(* CODESYS project Device.export

Project tree, tasks and I/O mapping:
  Device : CODESYS Control Win V3, 3S - Smart Software Solutions GmbH, version 3.5.17.30
    application Application
      libraries: Standard, * (System); CAA Memory, * (CAA Technical Workgroup); VisuDialogs, * (System); Standard64, * (System); VisuSymbols, 4.1.0.0 (System); Util, * (System); OwenTypes, 3.5.17.5 (Production association OWEN); Mx210 Assistant, 3.5.11.11 (Production association OWEN)
      task MainTask (cyclic, interval t#10ms, priority 1) calls PRG_Main, PRG_HMI
      task VISU_TASK (cyclic, interval 100 ms, priority 31) calls VisuElems.Visu_Prg
      data type E_LevelState
      data type E_WorkMode
      data type ST_ScheduleSlot
      global variables GVL_HMI
      global variables GVL_IO
      global variables GVL_Process
      global variables GVL_Schedules
      global variables TargetVars
      image pool ImagePool
      function block FB_AutoMode [ST]
      function block FB_LevelMonitor [ST]
      function block FB_ManualMode [ST]
      function block FB_Schedule [ST]
      program PRG_HMI [ST]
      program PRG_Main [ST]
      visualisation Visu_Levels
      visualisation Visu_Main
      visualisation Visu_Pumps
      visualisation Visu_Settings
      visualisation Visu_Valves
    Ethernet : Ethernet, 3S - Smart Software Solutions GmbH, version 3.5.17.0
      Modbus_TCP_Master : Modbus TCP Master, 3S - Smart Software Solutions GmbH, version 3.5.17.0
        MV210_214 : MV210-214, Production association OWEN, version 3.5.11.13
            input  Application.SA1_Auto : BOOL  // Битовая маска входов.Вход 1
            input  Application.SA2_Auto : BOOL  // Битовая маска входов.Вход 2
            input  Application.SA3_Auto : BOOL  // Битовая маска входов.Вход 3
            input  Application.SA4_Auto : BOOL  // Битовая маска входов.Вход 4
            input  Application.SA5_Auto : BOOL  // Битовая маска входов.Вход 5
            input  Application.SA6_Auto : BOOL  // Битовая маска входов.Вход 6
            input  Application.LVL_High : BOOL  // Битовая маска входов.Вход 7
            input  Application.LVL_Mid : BOOL  // Битовая маска входов.Вход 8
            input  Application.LVL_Low : BOOL  // Битовая маска входов.Вход 9
            input  Application.Flood : BOOL  // Битовая маска входов.Вход 10
            input  Application.SA7_Auto : BOOL  // Битовая маска входов.Вход 11
            input  Application.SA8_Manual : BOOL  // Битовая маска входов.Вход 12
            input  Application.SA9_Manual : BOOL  // Битовая маска входов.Вход 13
            input  Application.SA10_ManualOpen : BOOL  // Битовая маска входов.Вход 14
            input  Application.SA11_ManualOpen : BOOL  // Битовая маска входов.Вход 15
            input  Application.SA12_ManualOn : BOOL  // Битовая маска входов.Вход 16
            input  Application.SA13_Compressor : BOOL  // Битовая маска входов.Вход 17
            input  Application.DK_QF2 : BOOL  // Битовая маска входов.Вход 18
            input  Application.DK_QF3 : BOOL  // Битовая маска входов.Вход 19
            input  Application.DK_QF4 : BOOL  // Битовая маска входов.Вход 20
            input  Application.DK_QF5 : BOOL  // Битовая маска входов.Вход 21
            input  Application.DK_QF6 : BOOL  // Битовая маска входов.Вход 22
            input  Application.DK_QF7 : BOOL  // Битовая маска входов.Вход 23
            input  Application.DK_QF8 : BOOL  // Битовая маска входов.Вход 24
            input  Application.DK_QF9 : BOOL  // Битовая маска входов.Вход 25
            input  Application.DK_QF10 : BOOL  // Битовая маска входов.Вход 26
            input  Application.DK_QF11 : BOOL  // Битовая маска входов.Вход 27
            input  Application.DK_QF18 : BOOL  // Битовая маска входов.Вход 28
            input  Application.DK_QF19 : BOOL  // Битовая маска входов.Вход 29
            input  Application.DK_QF1 : BOOL  // Битовая маска входов.Вход 30
            unmapped channels: Tmp, Исключить модуль из опроса, Флаг ошибки, Битовая маска входов, Значение счетчика, Значение счетчика, Значение счетчика, Значение счетчика, Значение счетчика, Значение счетчика, Значение счетчика, Значение счетчика, Значение счетчика, Значение счетчика, Значение счетчика, Значение счетчика, Значение счетчика, Значение счетчика, Значение счетчика, Значение счетчика, Значение счетчика, Значение счетчика, Значение счетчика, Значение счетчика, Значение счетчика, Значение счетчика, Значение счетчика, Значение счетчика, Значение счетчика, Значение счетчика, Значение счетчика, Значение счетчика, Значение счетчика, Значение счетчика, Значение счетчика, Значение счетчика, Сбросить счетчик, Сбросить счетчик, Сбросить счетчик, Сбросить счетчик,
              Сбросить счетчик, Сбросить счетчик, Сбросить счетчик, Сбросить счетчик, Сбросить счетчик, Сбросить счетчик, Сбросить счетчик, Сбросить счетчик, Сбросить счетчик, Сбросить счетчик, Сбросить счетчик, Сбросить счетчик, Сбросить счетчик, Сбросить счетчик, Сбросить счетчик, Сбросить счетчик, Сбросить счетчик, Сбросить счетчик, Сбросить счетчик, Сбросить счетчик, Сбросить счетчик, Сбросить счетчик, Сбросить счетчик, Сбросить счетчик, Сбросить счетчик, Сбросить счетчик, Сбросить счетчик, Сбросить счетчик
        MV210_214_1 : MV210-214, Production association OWEN, version 3.5.11.13
            settings: Unit-ID = 2; IPAddress = [192, 168, 0, 2]
            input  Application.VFD1_Run : BOOL  // Битовая маска входов.Вход 1
            input  Application.VFD1_Alarm : BOOL  // Битовая маска входов.Вход 2
            input  Application.VFD2_Run : BOOL  // Битовая маска входов.Вход 3
            input  Application.VFD2_Alarm : BOOL  // Битовая маска входов.Вход 4
            input  Application.FB_KM0 : BOOL  // Битовая маска входов.Вход 5
            input  Application.FB_KM1 : BOOL  // Битовая маска входов.Вход 6
            input  Application.FB_KM2 : BOOL  // Битовая маска входов.Вход 7
            input  Application.FB_KM3 : BOOL  // Битовая маска входов.Вход 8
            input  Application.FB_KM4 : BOOL  // Битовая маска входов.Вход 9
            input  Application.FB_KM5 : BOOL  // Битовая маска входов.Вход 10
            input  Application.FB_KM5_1 : BOOL  // Битовая маска входов.Вход 11
            input  Application.FB_KM6 : BOOL  // Битовая маска входов.Вход 12
            input  Application.FB_KM6_1 : BOOL  // Битовая маска входов.Вход 13
            input  Application.FB_KM7 : BOOL  // Битовая маска входов.Вход 14
            input  Application.FB_KM8 : BOOL  // Битовая маска входов.Вход 15
            input  Application.FB_KM9 : BOOL  // Битовая маска входов.Вход 16
            input  Application.FB_KM10 : BOOL  // Битовая маска входов.Вход 17
            input  Application.FB_KM11 : BOOL  // Битовая маска входов.Вход 18
            input  Application.M2_Closed : BOOL  // Битовая маска входов.Вход 19
            input  Application.M2_Open : BOOL  // Битовая маска входов.Вход 20
            input  Application.M3_Closed : BOOL  // Битовая маска входов.Вход 21
            input  Application.M3_Open : BOOL  // Битовая маска входов.Вход 22
            input  Application.M4_Closed : BOOL  // Битовая маска входов.Вход 23
            input  Application.M4_Open : BOOL  // Битовая маска входов.Вход 24
            input  Application.M5_Closed : BOOL  // Битовая маска входов.Вход 25
            input  Application.M5_Open : BOOL  // Битовая маска входов.Вход 26
            unmapped channels: Tmp, Исключить модуль из опроса, Флаг ошибки, Битовая маска входов, Значение счетчика, Значение счетчика, Значение счетчика, Значение счетчика, Значение счетчика, Значение счетчика, Значение счетчика, Значение счетчика, Значение счетчика, Значение счетчика, Значение счетчика, Значение счетчика, Значение счетчика, Значение счетчика, Значение счетчика, Значение счетчика, Значение счетчика, Значение счетчика, Значение счетчика, Значение счетчика, Значение счетчика, Значение счетчика, Значение счетчика, Значение счетчика, Значение счетчика, Значение счетчика, Значение счетчика, Значение счетчика, Значение счетчика, Значение счетчика, Значение счетчика, Значение счетчика, Сбросить счетчик, Сбросить счетчик, Сбросить счетчик, Сбросить счетчик,
              Сбросить счетчик, Сбросить счетчик, Сбросить счетчик, Сбросить счетчик, Сбросить счетчик, Сбросить счетчик, Сбросить счетчик, Сбросить счетчик, Сбросить счетчик, Сбросить счетчик, Сбросить счетчик, Сбросить счетчик, Сбросить счетчик, Сбросить счетчик, Сбросить счетчик, Сбросить счетчик, Сбросить счетчик, Сбросить счетчик, Сбросить счетчик, Сбросить счетчик, Сбросить счетчик, Сбросить счетчик, Сбросить счетчик, Сбросить счетчик, Сбросить счетчик, Сбросить счетчик, Сбросить счетчик, Сбросить счетчик
        MU210_403 : MU210-403, Production association OWEN, version 3.5.11.13
            settings: Unit-ID = 3; IPAddress = [192, 168, 0, 3]
            output Application.CMD_KM0 : BOOL  // Битовая маска выходов (запись).Выход 1
            output Application.CMD_KM1 : BOOL  // Битовая маска выходов (запись).Выход 3
            output Application.CMD_KM2 : BOOL  // Битовая маска выходов (запись).Выход 4
            output Application.CMD_KM3 : BOOL  // Битовая маска выходов (запись).Выход 5
            output Application.CMD_KM4 : BOOL  // Битовая маска выходов (запись).Выход 6
            output Application.CMD_KM5_Close : BOOL  // Битовая маска выходов (запись).Выход 9
            output Application.CMD_KM5_1_Open : BOOL  // Битовая маска выходов (запись).Выход 10
            output Application.CMD_KM6_Close : BOOL  // Битовая маска выходов (запись).Выход 11
            output Application.CMD_KM6_1_Open : BOOL  // Битовая маска выходов (запись).Выход 12
            output Application.CMD_KM7 : BOOL  // Битовая маска выходов (запись).Выход 13
            output Application.CMD_KM8 : BOOL  // Битовая маска выходов (запись).Выход 14
            output Application.CMD_KM9 : BOOL  // Битовая маска выходов (запись).Выход 15
            output Application.CMD_KM10 : BOOL  // Битовая маска выходов (запись).Выход 16
            output Application.CMD_VFD1_Start : BOOL  // Битовая маска выходов (запись).Выход 17
            output Application.CMD_VFD1_Stop : BOOL  // Битовая маска выходов (запись).Выход 18
            output Application.CMD_VFD2_Start : BOOL  // Битовая маска выходов (запись).Выход 19
            output Application.CMD_VFD2_Stop : BOOL  // Битовая маска выходов (запись).Выход 20
            output Application.CMD_KM11_Light : BOOL  // Битовая маска выходов (запись).Выход 21
            unmapped channels: Tmp, Исключить модуль из опроса, Флаг ошибки, Битовая маска выходов (чтение), Битовая маска выходов (запись), Период ШИМ (чтение), Период ШИМ (чтение), Период ШИМ (чтение), Период ШИМ (чтение), Период ШИМ (чтение), Период ШИМ (чтение), Период ШИМ (чтение), Период ШИМ (чтение), Период ШИМ (чтение), Период ШИМ (чтение), Период ШИМ (чтение), Период ШИМ (чтение), Период ШИМ (чтение), Период ШИМ (чтение), Период ШИМ (чтение), Период ШИМ (чтение), Период ШИМ (чтение), Период ШИМ (чтение), Период ШИМ (чтение), Период ШИМ (чтение), Период ШИМ (чтение), Период ШИМ (чтение), Период ШИМ (чтение), Период ШИМ (чтение), Период ШИМ (запись), Период ШИМ (запись), Период ШИМ (запись), Период ШИМ (запись), Период ШИМ (запись), Период ШИМ (запись), Период ШИМ (запись), Период ШИМ (запись), Период ШИМ (запись), Период ШИМ (запись), Период ШИМ (запись),
              Период ШИМ (запись), Период ШИМ (запись), Период ШИМ (запись), Период ШИМ (запись), Период ШИМ (запись), Период ШИМ (запись), Период ШИМ (запись), Период ШИМ (запись), Период ШИМ (запись), Период ШИМ (запись), Период ШИМ (запись), Период ШИМ (запись), Период ШИМ (запись), Коэффициент заполнения ШИМ (чтение), Коэффициент заполнения ШИМ (чтение), Коэффициент заполнения ШИМ (чтение), Коэффициент заполнения ШИМ (чтение), Коэффициент заполнения ШИМ (чтение), Коэффициент заполнения ШИМ (чтение), Коэффициент заполнения ШИМ (чтение), Коэффициент заполнения ШИМ (чтение), Коэффициент заполнения ШИМ (чтение), Коэффициент заполнения ШИМ (чтение), Коэффициент заполнения ШИМ (чтение), Коэффициент заполнения ШИМ (чтение), Коэффициент заполнения ШИМ (чтение), Коэффициент заполнения ШИМ (чтение), Коэффициент заполнения ШИМ (чтение), Коэффициент заполнения ШИМ (чтение), Коэффициент заполнения ШИМ (чтение), Коэффициент заполнения ШИМ (чтение), Коэффициент заполнения ШИМ (чтение), Коэффициент заполнения ШИМ (чтение), Коэффициент заполнения ШИМ (чтение), Коэффициент заполнения ШИМ (чтение), Коэффициент заполнения ШИМ (чтение), Коэффициент заполнения ШИМ (чтение), Коэффициент заполнения ШИМ (запись), Коэффициент заполнения ШИМ (запись), Коэффициент заполнения ШИМ (запись),
              Коэффициент заполнения ШИМ (запись), Коэффициент заполнения ШИМ (запись), Коэффициент заполнения ШИМ (запись), Коэффициент заполнения ШИМ (запись), Коэффициент заполнения ШИМ (запись), Коэффициент заполнения ШИМ (запись), Коэффициент заполнения ШИМ (запись), Коэффициент заполнения ШИМ (запись), Коэффициент заполнения ШИМ (запись), Коэффициент заполнения ШИМ (запись), Коэффициент заполнения ШИМ (запись), Коэффициент заполнения ШИМ (запись), Коэффициент заполнения ШИМ (запись), Коэффициент заполнения ШИМ (запись), Коэффициент заполнения ШИМ (запись), Коэффициент заполнения ШИМ (запись), Коэффициент заполнения ШИМ (запись), Коэффициент заполнения ШИМ (запись), Коэффициент заполнения ШИМ (запись), Коэффициент заполнения ШИМ (запись), Коэффициент заполнения ШИМ (запись)
        MU210_502 : MU210-502, Production association OWEN, version 3.5.11.13
            settings: Unit-ID = 4; IPAddress = [192, 168, 0, 4]
            output Application.VFD1_SpeedCmd : localTypes:OutputValue  // Значение выхода (запись)
            output Application.VFD2_SpeedCmd : localTypes:OutputValue  // Значение выхода (запись)
            unmapped channels: Tmp, Исключить модуль из опроса, Флаг ошибки, Битовая маска диагностики выходов, Значение выхода (чтение), Значение выхода (чтение), Значение выхода (чтение), Значение выхода (чтение), Значение выхода (чтение), Значение выхода (чтение), Значение выхода (запись), Значение выхода (запись), Значение выхода (запись), Значение выхода (запись), Код статуса, Код статуса, Код статуса, Код статуса, Код статуса, Код статуса, Температура модуля, Перегрев модуля
  5ce3da45-db07-42e7-a21c-a00fff4ed8f6|PLC_Project\HMI\svg\Visu_Alarm_banner.svg
  5ce3da45-db07-42e7-a21c-a00fff4ed8f6|PLC_Project\HMI\svg\Visu_Levels_bg.svg
  5ce3da45-db07-42e7-a21c-a00fff4ed8f6|PLC_Project\HMI\svg\Visu_Main_bg.svg
  5ce3da45-db07-42e7-a21c-a00fff4ed8f6|PLC_Project\HMI\svg\Visu_Pumps_bg.svg
  5ce3da45-db07-42e7-a21c-a00fff4ed8f6|PLC_Project\HMI\svg\Visu_Settings_bg.svg
  5ce3da45-db07-42e7-a21c-a00fff4ed8f6|PLC_Project\HMI\svg\Visu_Valves_bg.svg
*)

// Device/Application/E_LevelState
(* Имена LEV_* — не LVL_*: в CODESYS идентификаторы без учёта регистра,
   LVL_HIGH совпадает с BOOL LVL_High из GVL_IO → ошибка C0066/C0231 *)
TYPE E_LevelState :
(
    LEV_EMPTY := 0,
    LEV_LOW   := 1,
    LEV_MID   := 2,
    LEV_HIGH  := 3,
    LEV_FAULT := 4
);
END_TYPE

// Device/Application/E_WorkMode
TYPE E_WorkMode :
(
    MODE_MANUAL := 0,
    MODE_AUTO   := 1
);
END_TYPE

// Device/Application/ST_ScheduleSlot
TYPE ST_ScheduleSlot :
STRUCT
    Enable    : BOOL;
    StartHour : BYTE;
    StartMin  : BYTE;
    StopHour  : BYTE;
    StopMin   : BYTE;
END_STRUCT
END_TYPE

// Device/Application/GVL_HMI
VAR_GLOBAL
    // --- Управление с HMI (только в автомате, если не ручной ключ на щите) ---
    HMI_AutoEnable     : BOOL := TRUE;
    HMI_ResetAlarm     : BOOL;
    HMI_LightOn        : BOOL;
    HMI_FillValveForce : BOOL;
    HMI_Page           : INT := 0;   // 0=главная, 1=насосы, 2=краны, 3=уровни, 4=настройки

    // --- Статусы системы ---
    Status_Ready       : BOOL;
    Status_Running     : BOOL;
    Status_Alarm       : BOOL;
    Status_Manual      : BOOL;
    Status_FillPhase   : BOOL;
    Disp_LevelPct      : INT;
    Disp_LevelText     : STRING[20];

    // --- Аварии ---
    Alarm_DryRun       : BOOL;
    Alarm_Flood        : BOOL;
    Alarm_VFD1         : BOOL;
    Alarm_VFD2         : BOOL;
    Alarm_AnyDK        : BOOL;

    // --- Насосы Н1-Н6, М1 (работа = команда AND обратная связь где есть) ---
    Disp_N1_Run        : BOOL;
    Disp_N2_Run        : BOOL;
    Disp_N3_Run        : BOOL;
    Disp_N4_Run        : BOOL;
    Disp_N5_Run        : BOOL;
    Disp_N6_Run        : BOOL;
    Disp_M1_Run        : BOOL;
    Disp_N1_Manual     : BOOL;
    Disp_N2_Manual     : BOOL;
    Disp_N3_Manual     : BOOL;
    Disp_N4_Manual     : BOOL;
    Disp_N5_Manual     : BOOL;
    Disp_N6_Manual     : BOOL;
    Disp_M1_Manual     : BOOL;
    Disp_N1_Alarm      : BOOL;
    Disp_N3_Alarm      : BOOL;

    // --- Краны и прочее ---
    Disp_M2_Open       : BOOL;
    Disp_M3_Open       : BOOL;
    Disp_M4_Open       : BOOL;
    Disp_M5_Open       : BOOL;
    Disp_UF_On         : BOOL;
    Disp_Compressor    : BOOL;
    Disp_Light         : BOOL;

    // --- Уровни (дискрет) ---
    Disp_LvlHigh       : BOOL;
    Disp_LvlMid        : BOOL;
    Disp_LvlLow        : BOOL;
    Disp_Flood         : BOOL;

    // --- Время для расписания (из RTC, заполняется в PRG_HMI) ---
    HMI_NowHour        : BYTE;
    HMI_NowMin         : BYTE;
    HMI_NowSec         : BYTE;
	
	Col_OK : DWORD := 16#00B6C42E;
    Col_Manual : DWORD := 16#006AC4E9;
    Col_ModeBg : DWORD;
	ModeText : STRING[10];
	Disp_TimeText : STRING[8];

END_VAR

// Device/Application/GVL_IO
(* GVL_IO — входы/выходы щита ЩУ, СПК210-07-CS *)
VAR_GLOBAL
    (* Ключи SA: TRUE = автомат *)
    SA1_Auto, SA2_Auto, SA3_Auto, SA4_Auto, SA5_Auto, SA6_Auto : BOOL;
    SA7_Auto : BOOL;
    SA8_Manual, SA9_Manual : BOOL;
    SA8_1_Open, SA8_1_Close, SA9_1_Open, SA9_1_Close : BOOL;
    SA10_ManualOpen, SA11_ManualOpen, SA12_ManualOn, SA13_Compressor : BOOL;
    SA14_LightManual : BOOL;

    (* Уровни и затопление — XT4, KL4 *)
    LVL_High, LVL_Mid, LVL_Low, Flood : BOOL;

    (* Контакты доп. защиты автоматов QF (ДК), лист 6 схемы *)
    (* QF12–QF17 на схему не выведены — переменные не используются *)
    DK_QF1, DK_QF2, DK_QF3, DK_QF4, DK_QF5, DK_QF6 : BOOL;
    DK_QF7, DK_QF8, DK_QF9, DK_QF10, DK_QF11 : BOOL;
    DK_QF18, DK_QF19 : BOOL;

    (* УПП и обратная связь пускателей — MV210-214 A4 *)
    VFD1_Run, VFD1_Alarm, VFD2_Run, VFD2_Alarm : BOOL;
    
    (* Аналоговое задание скорости на УПП — модуль MU210-502 (AO1/AO2), 4–20 mA по схеме *)
    (* Тип UINT выбран, чтобы совпасть с типом канала AO в описании устройства и убрать предупреждение REAL→UINT. *)
    VFD1_SpeedCmd, VFD2_SpeedCmd : UINT;
    FB_KM0, FB_KM1, FB_KM2, FB_KM3, FB_KM4 : BOOL;
    FB_KM5, FB_KM5_1, FB_KM6, FB_KM6_1 : BOOL;
    FB_KM7, FB_KM8, FB_KM9, FB_KM10, FB_KM11 : BOOL;

    (* Концевики кранов XT5 *)
    M2_Closed, M2_Open, M3_Closed, M3_Open : BOOL;
    M4_Closed, M4_Open, M5_Closed, M5_Open : BOOL;
END_VAR

VAR_GLOBAL
    (* Команды на выходы MU210-403 *)
    CMD_KM0, CMD_KM1, CMD_KM2, CMD_KM3, CMD_KM4 : BOOL;
    CMD_KM5_Close, CMD_KM5_1_Open, CMD_KM6_Close, CMD_KM6_1_Open : BOOL;
    CMD_KM7, CMD_KM8, CMD_KM9, CMD_KM10, CMD_KM11_Light : BOOL;
    CMD_VFD1_Start, CMD_VFD1_Stop, CMD_VFD2_Start, CMD_VFD2_Stop : BOOL;
END_VAR

// Device/Application/GVL_Process
VAR_GLOBAL RETAIN
    WorkMode           : E_WorkMode := MODE_AUTO;
    SystemReady        : BOOL;
    SystemRunning      : BOOL;
    GlobalStop         : BOOL;
    Alarm_Active       : BOOL;
    Alarm_DryRun       : BOOL;
    Alarm_Flood        : BOOL;
    FillPhaseDone      : BOOL;
    LightTimerPreset   : TIME := T#30M;
    VFD_Speed_RunPct   : UINT := 1000;  (* MU210-502: 0…1000 соответствует 0…100% *)
END_VAR

// Device/Application/GVL_Schedules
VAR_GLOBAL RETAIN
    Sched_N1, Sched_N2, Sched_N3, Sched_N4, Sched_N5, Sched_N6, Sched_M1 : ST_ScheduleSlot;
END_VAR

// Device/Application/TargetVars
{attribute 'qualified_only'}
VAR_GLOBAL
	stBuzzer:	 	OwenTypes.TRG_Buzzer;
	stDebug: 	 	OwenTypes.TRG_Debug;
	stDrives: 	 	OwenTypes.TRG_Drives;
	stRtc:		 	OwenTypes.TRG_RTC;
	stOwenCloud:	OwenTypes.TRG_OwenCloud;
	stInfo:		 	OwenTypes.TRG_Info;
	stWatchdog:	 	OwenTypes.TRG_Watchdog;
	stNetwork:		OwenTypes.TRG_Network;
	stScreen:		OwenTypes.TRG_Screen;
END_VAR

// Device/Application/PRG_Main
PROGRAM PRG_Main
VAR
    LevelMon : FB_LevelMonitor;
    Manual   : FB_ManualMode;
    Auto     : FB_AutoMode;
    i : INT;
END_VAR

LevelMon(High := GVL_IO.LVL_HIGH, Mid := LVL_Mid, Low := LVL_Low, Flood := Flood);

// Определение общего режима: если любой SA в ручном — приоритет ручного для этой группы
WorkMode := MODE_AUTO;
IF NOT SA1_Auto OR NOT SA2_Auto OR NOT SA3_Auto OR NOT SA4_Auto OR NOT SA5_Auto OR NOT SA6_Auto OR NOT SA7_Auto THEN
    WorkMode := MODE_MANUAL;
END_IF

// Сброс аварии
IF HMI_ResetAlarm THEN
    GlobalStop := FALSE;
    GVL_Process.Alarm_Active := FALSE;
    GVL_Process.Alarm_DryRun := FALSE;
    GVL_Process.Alarm_Flood := FALSE;
END_IF

CASE WorkMode OF
    MODE_MANUAL:
        Manual(Enable := TRUE);
    MODE_AUTO:
        IF HMI_AutoEnable THEN
            Auto(
                Enable := TRUE,
                LevelState := LevelMon.State,
                LevelAllowRun := LevelMon.AllowRun,
                LevelNeedFill := LevelMon.NeedFill,
                LevelEmergencyStop := LevelMon.EmergencyStop
            );
        END_IF
END_CASE

// Задание скорости на УПП (MU210-502 AO): 0% — стоп, VFD_Speed_RunPct (100%) — при пуске
VFD1_SpeedCmd := SEL(CMD_VFD1_Start AND NOT GlobalStop, UINT#0, VFD_Speed_RunPct);
VFD2_SpeedCmd := SEL(CMD_VFD2_Start AND NOT GlobalStop, UINT#0, VFD_Speed_RunPct);

END_PROGRAM

// Device/Application/FB_LevelMonitor
FUNCTION_BLOCK FB_LevelMonitor
VAR_INPUT
    High, Mid, Low, Flood : BOOL;
END_VAR
VAR_OUTPUT
    State : E_LevelState;
    AllowRun : BOOL;
    NeedFill : BOOL;
    EmergencyStop : BOOL;
END_VAR

IF Flood OR Low THEN
    State := LEV_FAULT;
    AllowRun := FALSE;
    NeedFill := FALSE;
    EmergencyStop := TRUE;
ELSIF High THEN
    State := LEV_HIGH;
    AllowRun := TRUE;
    NeedFill := FALSE;
    EmergencyStop := FALSE;
ELSIF Mid THEN
    State := LEV_MID;
    AllowRun := TRUE;
    NeedFill := FALSE;
    EmergencyStop := FALSE;
ELSE
    State := LEV_LOW;
    AllowRun := FALSE;
    NeedFill := TRUE;
    EmergencyStop := FALSE;
END_IF

END_FUNCTION_BLOCK

// Device/Application/FB_ManualMode
FUNCTION_BLOCK FB_ManualMode
VAR_INPUT
    Enable : BOOL;
END_VAR
VAR_OUTPUT
    AnyManualActive : BOOL;
END_VAR

// Ручной режим: прямое управление ключами, без защит сухого хода
IF NOT Enable THEN
    AnyManualActive := FALSE;
    RETURN;
END_IF

// Н1 через УПП — при SA1 в ручном включаем пуск (без interlock)
IF NOT SA1_Auto THEN
    CMD_VFD1_Start := TRUE;
    CMD_VFD1_Stop := FALSE;
ELSE
    CMD_VFD1_Start := FALSE;
END_IF

IF NOT SA2_Auto THEN CMD_KM1 := TRUE; END_IF  // Н4 — KM1 на схеме для фильтра
IF NOT SA3_Auto THEN CMD_VFD2_Start := TRUE; END_IF
IF NOT SA4_Auto THEN CMD_KM1 := TRUE; END_IF
IF NOT SA5_Auto THEN CMD_KM2 := TRUE; END_IF
IF NOT SA6_Auto THEN CMD_KM3 := TRUE; END_IF
IF NOT SA7_Auto THEN CMD_KM0 := TRUE; END_IF

// M2/M3 — SA8.1/SA9.1 открыть/закрыть
IF SA8_Manual THEN
    CMD_KM5_Close := SA8_1_Close;
    CMD_KM5_1_Open := SA8_1_Open;
END_IF
IF SA9_Manual THEN
    CMD_KM6_Close := SA9_1_Close;
    CMD_KM6_1_Open := SA9_1_Open;
END_IF

// M4/M5 — при ручном сразу открыты, при 0 закрыты
IF SA10_ManualOpen THEN CMD_KM7 := TRUE; ELSE CMD_KM7 := FALSE; END_IF
IF SA11_ManualOpen THEN CMD_KM8 := TRUE; ELSE CMD_KM8 := FALSE; END_IF

IF SA12_ManualOn THEN CMD_KM9 := TRUE; ELSE CMD_KM9 := FALSE; END_IF
CMD_KM10 := SA13_Compressor;  // только ручной
CMD_KM11_Light := SA14_LightManual;

AnyManualActive := NOT SA1_Auto OR NOT SA2_Auto OR NOT SA3_Auto OR NOT SA4_Auto
    OR NOT SA5_Auto OR NOT SA6_Auto OR NOT SA7_Auto OR SA8_Manual OR SA9_Manual
    OR SA10_ManualOpen OR SA11_ManualOpen OR SA12_ManualOn OR SA13_Compressor;

END_FUNCTION_BLOCK

// Device/Application/FB_AutoMode
FUNCTION_BLOCK FB_AutoMode
VAR_INPUT
    Enable : BOOL;
    LevelState : E_LevelState;
    LevelAllowRun : BOOL;
    LevelNeedFill : BOOL;
    LevelEmergencyStop : BOOL;
END_VAR
VAR
    SchN1, SchN2, SchN3, SchN4, SchN5, SchN6, SchM1 : FB_Schedule;
    NowHour, NowMin : BYTE;
    LightTimer : TON;
END_VAR

IF NOT Enable THEN RETURN; END_IF

// Аварийная остановка
IF LevelEmergencyStop THEN
    GlobalStop := TRUE;
    Alarm_Active := TRUE;
    GVL_Process.Alarm_DryRun := LVL_Low AND NOT Flood;
    GVL_Process.Alarm_Flood := Flood;
    RETURN;
END_IF

// Фаза наполнения: ждём верхний уровень
// Верхний уровень: LEV_HIGH (enum), дискрет DI — LVL_High (BOOL), имена разные!
IF NOT FillPhaseDone THEN
    IF LevelState = LEV_HIGH THEN
        FillPhaseDone := TRUE;
        SystemReady := TRUE;
    ELSE
        // Долив M4 при необходимости
        CMD_KM7 := LevelNeedFill OR HMI_FillValveForce;
        SystemRunning := CMD_KM7;
        RETURN;
    END_IF
END_IF

// Рабочий режим между средним и нижним
IF LevelState = LEV_FAULT THEN
    GlobalStop := TRUE;
    RETURN;
END_IF

SystemRunning := LevelAllowRun;

// Расписания (заглушки — настраиваются в GVL_Schedules RETAIN)
SchN1(Enable := SA1_Auto, Slot := Sched_N1, NowHour := NowHour, NowMin := NowMin);
CMD_VFD1_Start := SchN1.Active AND LevelAllowRun AND NOT VFD1_Alarm;
CMD_VFD1_Stop := NOT SchN1.Active OR GlobalStop;

SchN3(Enable := SA3_Auto, Slot := Sched_N3, NowHour := NowHour, NowMin := NowMin);
CMD_VFD2_Start := SchN3.Active AND LevelAllowRun AND NOT VFD2_Alarm;

SchN4(Enable := SA4_Auto, Slot := Sched_N4, NowHour := NowHour, NowMin := NowMin);
CMD_KM1 := SchN4.Active AND LevelAllowRun;

SchN5(Enable := SA5_Auto, Slot := Sched_N5, NowHour := NowHour, NowMin := NowMin);
CMD_KM2 := SchN5.Active AND LevelAllowRun;

SchN6(Enable := SA6_Auto, Slot := Sched_N6, NowHour := NowHour, NowMin := NowMin);
CMD_KM3 := SchN6.Active AND LevelAllowRun;

SchM1(Enable := SA7_Auto, Slot := Sched_M1, NowHour := NowHour, NowMin := NowMin);
CMD_KM0 := SchM1.Active AND LevelAllowRun;

// M4 долив по 3 уровням в авто
CMD_KM7 := LevelNeedFill AND NOT SA10_ManualOpen;

// M5 по затоплению — открыть при Flood, иначе закрыть
CMD_KM8 := Flood;

// M2/M3 — требуется уточнение заказчиком: по умолчанию открыты при работе
IF SystemRunning THEN
    CMD_KM5_1_Open := TRUE;
    CMD_KM6_1_Open := TRUE;
END_IF

// Подсветка по таймеру
LightTimer(IN := SystemRunning, PT := LightTimerPreset);
CMD_KM11_Light := LightTimer.Q OR HMI_LightOn;

END_FUNCTION_BLOCK

// Device/Application/FB_Schedule
FUNCTION_BLOCK FB_Schedule
VAR_INPUT
    Enable : BOOL;
    Slot : ST_ScheduleSlot;
    NowHour, NowMin : BYTE;
END_VAR
VAR_OUTPUT
    Active : BOOL;
END_VAR
VAR
    tStart, tStop, tNow : TIME;
END_VAR

IF NOT Enable OR NOT Slot.Enable THEN
    Active := FALSE;
    RETURN;
END_IF
tStart := (T#1H * Slot.StartHour) + (T#1M * Slot.StartMin);
tStop  := (T#1H * Slot.StopHour)  + (T#1M * Slot.StopMin);
tNow   := (T#1H * NowHour) + (T#1M * NowMin);
IF tStart <= tStop THEN
    Active := (tNow >= tStart) AND (tNow < tStop);
ELSE
    Active := (tNow >= tStart) OR (tNow < tStop);
END_IF

END_FUNCTION_BLOCK

// Device/Application/PRG_HMI
PROGRAM PRG_HMI
VAR
    lvlText : STRING[20];
END_VAR


// Время (OwenRTC — при наличии привязать к SysTime; иначе заглушка)
// HMI_NowHour := ...  — настраивается через OwenRTC в Device Tree

Status_Manual := (WorkMode = MODE_MANUAL);
Status_FillPhase := NOT FillPhaseDone AND (WorkMode = MODE_AUTO);

Disp_LvlHigh := LVL_High;
Disp_LvlMid  := LVL_Mid;
Disp_LvlLow  := LVL_Low;
Disp_Flood   := Flood;

// Owen: CASE только с целочисленным селектором, не CASE TRUE OF с BOOL
IF Flood THEN
    lvlText := 'Затопление';
ELSIF LVL_High THEN
    lvlText := 'Верхний';
ELSIF LVL_Mid THEN
    lvlText := 'Рабочий';
ELSIF LVL_Low THEN
    lvlText := 'Нижний';
ELSE
    lvlText := 'Нет данных';
END_IF
Disp_LevelText := lvlText;

// Насосы
Disp_N1_Manual := NOT SA1_Auto;
Disp_N2_Manual := NOT SA2_Auto;
Disp_N3_Manual := NOT SA3_Auto;
Disp_N4_Manual := NOT SA4_Auto;
Disp_N5_Manual := NOT SA5_Auto;
Disp_N6_Manual := NOT SA6_Auto;
Disp_M1_Manual := NOT SA7_Auto;

Disp_N1_Run := CMD_VFD1_Start OR VFD1_Run;
Disp_N2_Run := FALSE;  // Н2 — прямой пуск, добавить FB при появлении DI
Disp_N3_Run := CMD_VFD2_Start OR VFD2_Run;
Disp_N4_Run := CMD_KM1 OR FB_KM1;
Disp_N5_Run := CMD_KM2 OR FB_KM2;
Disp_N6_Run := CMD_KM3 OR FB_KM3;
Disp_M1_Run := CMD_KM0 OR FB_KM0;
Disp_N1_Alarm := VFD1_Alarm;
Disp_N3_Alarm := VFD2_Alarm;

// Краны
Disp_M2_Open := CMD_KM5_1_Open OR M2_Open;
Disp_M3_Open := CMD_KM6_1_Open OR M3_Open;
Disp_M4_Open := CMD_KM7 OR M4_Open;
Disp_M5_Open := CMD_KM8 OR M5_Open;
Disp_UF_On := CMD_KM9 OR FB_KM9;
Disp_Compressor := CMD_KM10 OR FB_KM10;
Disp_Light := CMD_KM11_Light OR FB_KM11;

Alarm_VFD1 := VFD1_Alarm;
Alarm_VFD2 := VFD2_Alarm;
// Имена в GVL_HMI и GVL_Process совпадают — указывать GVL явно
GVL_HMI.Alarm_DryRun := GVL_Process.Alarm_DryRun;
GVL_HMI.Alarm_Flood := GVL_Process.Alarm_Flood;
Alarm_AnyDK := DK_QF1 OR DK_QF2 OR DK_QF3 OR DK_QF4 OR DK_QF5 OR DK_QF6 OR DK_QF7
    OR DK_QF8 OR DK_QF9 OR DK_QF10 OR DK_QF11 OR DK_QF18 OR DK_QF19;

Status_Ready := SystemReady;
Status_Running := SystemRunning;
Status_Alarm := NOT GVL_Process.Alarm_Active;

// Owen: SEL(G,…) здесь G=BOOL не всегда принимается — через IF
IF LVL_High THEN
    Disp_LevelPct := 100;
ELSIF LVL_Mid THEN
    Disp_LevelPct := 60;
ELSIF LVL_Low THEN
    Disp_LevelPct := 20;
ELSE
    Disp_LevelPct := 0;
END_IF

IF GVL_HMI.Status_Manual THEN
    GVL_HMI.Col_ModeBg := GVL_HMI.Col_Manual;
ELSE
    GVL_HMI.Col_ModeBg := GVL_HMI.Col_OK;
END_IF

IF GVL_HMI.Status_Manual THEN
    GVL_HMI.ModeText := 'Ручной';
ELSE
    GVL_HMI.ModeText := 'Автомат';
END_IF

GVL_HMI.Disp_TimeText :=
    CONCAT(CONCAT(BYTE_TO_STRING(GVL_HMI.HMI_NowHour), ':'), BYTE_TO_STRING(GVL_HMI.HMI_NowMin));

END_PROGRAM

// Device/Application/Visu_Levels
VISUALIZATION Visu_Levels  // 800x480, background image ImagePool.Visu_Levels_bg
END_VISUALIZATION

// Device/Application/Visu_Main
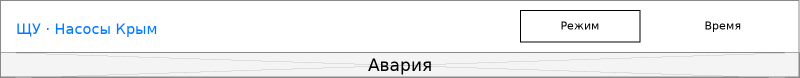
VISUALIZATION Visu_Main  // 800x78, background image ImagePool.Visu_Main_bg
    Label (12,14 150x30), "ЩУ · Насосы Крым"
    RoundedRectangle (520,10 120x32), "Режим", text variable: ModeText, colour variable: Col_ModeBg
    Textfield (648,11 150x30), "Время", text variable: Disp_TimeText
    Image (0,52 800x26), "Авария", invisible if: Status_Alarm, image: ImagePool.Visu_Alarm_banner
END_VISUALIZATION

// Device/Application/Visu_Pumps
VISUALIZATION Visu_Pumps  // 2x2, background image ImagePool.Visu_Pumps_bg
END_VISUALIZATION

// Device/Application/Visu_Settings
VISUALIZATION Visu_Settings  // 2x2, background image ImagePool.Visu_Settings_bg
END_VISUALIZATION

// Device/Application/Visu_Valves
VISUALIZATION Visu_Valves  // 2x2, background image ImagePool.Visu_Valves_bg
END_VISUALIZATION
